# EPICS autosave request: ADPICam/iocs/PICamIOC/iocBoot/iocPICam/auto_settings.req
file "PICam_settings.req",        P=$(P),  R=cam1:
file "NDStdArrays_settings.req",  P=$(P),  R=image1:
file "commonPlugin_settings.req", P=$(P)
